TYPE ST_TxRxQueue :
STRUCT
	txCounter : UINT;
	rxCounter : UINT;
	noOfMessages : UINT;
	messages : ARRAY[0..9] OF ST_TxRxMessage;
END_STRUCT
END_TYPE

(* stored: Version 1.1.0.1, ProductVersion 3.1.4024.9
   DUT ST_TxRxQueue: Id {0847a097-abb9-451c-a740-4a75d5ebc653} *)
